FUNCTION WRITE_PROTECTED_TIME_OF_DAY
VAR_INPUT
    Ptr : POINTER TO TIME_OF_DAY;
    Value : TIME_OF_DAY;
END_VAR

Ptr^ := Value;

END_FUNCTION

(* stored: Version 1.1.0.1
   POU WRITE_PROTECTED_TIME_OF_DAY: Id {c9020a0a-7555-43c0-b5e9-58aed910df89}, SpecialFunc None *)
